{attribute 'GeneratedUsingTerminal: EP7402-0057-0017'}
{attribute addProperty BoxType "EP7402-0057-0017"}
{attribute addProperty Id "Info_dataAT %I*ARRAY[0..2] OF UINT6"}
{attribute addProperty CRC "1532541242"}
{attribute addProperty Size "6"}
TYPE STM_Synchron_info_data_Channel_DD535D91 :
STRUCT
	{attribute addProperty Name "Info_data"}
	Info_data AT %I* : ARRAY[0..2] OF UINT;
END_STRUCT
END_TYPE

(* stored: Version 1.2.0.0, ProductVersion 3.1.4024.9
   DUT STM_Synchron_info_data_Channel_DD535D91: Id {681f967f-4680-4995-93b4-809f84bc65de} *)
